FUNCTION TFPalletizerPickRollerPriority : uINT (*Restituisce il numero del Pick-Point Sul quale deve può essere effettuato il prelievo*)
VAR_INPUT
	WorkArea 					: POINTER TO ARRAY [1..MAXAREA] OF TFMachinePalletizer_WorkArea;
	WorkAreaState 				: POINTER TO ARRAY [1..MAXAREA] OF TFMachinePalletizer_WorkAreaState;
	LastRequetsID : string;	(* Codice univoco ultimo prodotto scaricato *)
	Abilita_Priorita_Impostata_Da_Rulliere : BOOL;	(* Se TRUE la priorità del prelievo è gestita della rulliere *)
	//Priorita_Avanzata_Abilitata	: BOOL;					(* Se TRUE la priorità del prelievo è gestita in modo ottimale, 
	//												 	cerco di completare la postazione più completa *) 		
	
END_VAR
VAR
	wpp : UINT;
	pc : INT;
	WPP_Ordinati_Per_Priorita : ARRAY[1..MAXAREA] OF UINT;
	Indice_WPP_Ordinati : ARRAY[1..MAXAREA] OF UINT;
	Indice_Tmp : UINT;
	i	: UINT;
END_VAR

(* Ordinamento in ordine decrescente di Priorità.. in questo modo si cerca la disponibilità sulla rulliera con priorià più alta *)
IF Abilita_Priorita_Impostata_Da_Rulliere THEN
	FOR i := 1 TO MAXAREAPRESENT DO
		WPP_Ordinati_Per_Priorita[i] := INT_TO_UINT(WorkAreaState^[i].TransportState.Priority);
		Indice_WPP_Ordinati[i] := i;
	END_FOR	
	FOR wpp:= 1 TO MAXAREAPRESENT DO 
		IF WPP_Ordinati_Per_Priorita[wpp] <= WPP_Ordinati_Per_Priorita[wpp+1] THEN
			Indice_Tmp := Indice_WPP_Ordinati[wpp];
			Indice_WPP_Ordinati[wpp] := wpp + 1;
 			Indice_WPP_Ordinati[wpp+1] := Indice_Tmp;
			wpp := 1;
		END_IF
	END_FOR
END_IF
(* Per tutte le WorkPickPoint Attive *)
FOR wpp := 1 TO MAXAREAPRESENT DO
	IF WorkArea^[Indice_WPP_Ordinati[wpp]].Enable = 1 THEN
		(* Verifico disponibilità Lastra *)
		IF WorkAreaState^[Indice_WPP_Ordinati[wpp]].TransportState.State = WORKPICKPOINT_STATE_AUTO THEN
			IF WorkAreaState^[Indice_WPP_Ordinati[wpp]].TransportState.ProdPresence = WORKPICKPOINT_PRODOTTO_PRESENTE THEN
				(* Verifico se il codice è giusto *)
				IF WorkAreaState^[Indice_WPP_Ordinati[wpp]].TransportState.DataElement.WorkingID = LastRequetsID AND LastRequetsID <> '' THEN
					TFPalletizerPickRollerPriority := (Indice_WPP_Ordinati[wpp]);
					RETURN;
				ELSE
					;//Proseguo
				END_IF
			END_IF
		END_IF
	END_IF
END_FOR
TFPalletizerPickRollerPriority := 1;//Nel caso non abbia trovato nulla metto la postazione 1 come postazione di Default

END_FUNCTION

(* stored: Version 1.1.0.1, ProductVersion 3.1.4024.11
   POU TFPalletizerPickRollerPriority: Id {9eb9d089-0bdf-4384-82b3-bfbb894d467f}, SpecialFunc None *)
